(* CoDeSys 2.3.9.37 project: Cap6_10.pro *)
(* Libraries: Standard.LIB 4.10.05 12:14:46 *)

(* Global variable list: Global_Variables *)
VAR_GLOBAL

(* Entradas *)
     A:BOOL;
     B:BOOL;
     Encendido:BOOL;

(*Salidas *)
  Bomba1:BOOL;
  Bomba2:BOOL;

END_VAR

(* POU PLC_PRG, ST *)
PROGRAM PLC_PRG
VAR

END_VAR
Control();
Simulacion();
END_PROGRAM

(* POU Control, LD *)
PROGRAM Control
VAR
END_VAR
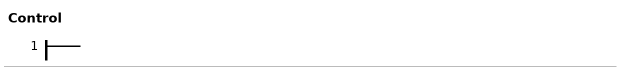
_LD_ (* Ladder Diagram *)
NETWORK 1
	*
_END_LD_
(* the same logic as Structured Text *)
(* Network 1 *)
END_PROGRAM

(* POU Simulacion, ST *)
PROGRAM Simulacion
VAR
   posy:INT;
	PrimerCiclo: BOOL:=TRUE;
	posInicial: INT;
END_VAR
IF posy>-187 THEN
IF (Bomba1=TRUE AND Bomba2=TRUE) THEN
  posy:=posy-2;
ELSE
     IF (Bomba1=TRUE OR Bomba2=TRUE) THEN
            posy:=posy-1;
     END_IF
END_IF
END_IF

IF (Bomba1=FALSE AND Bomba2=FALSE) THEN
IF posy<52 THEN
  posy:=posy+1;
END_IF
END_IF



IF posy<-50 THEN
  A:=TRUE;
ELSE
  A:=FALSE;
END_IF

IF posy<=-164 THEN
  B:=TRUE;
ELSE
  B:=FALSE;
END_IF

(* Solo en primer ciclo*)
IF (PrimerCiclo) THEN
    PrimerCiclo:=FALSE;
    posy:=posInicial;
END_IF
END_PROGRAM

(* Visualisation Deposito
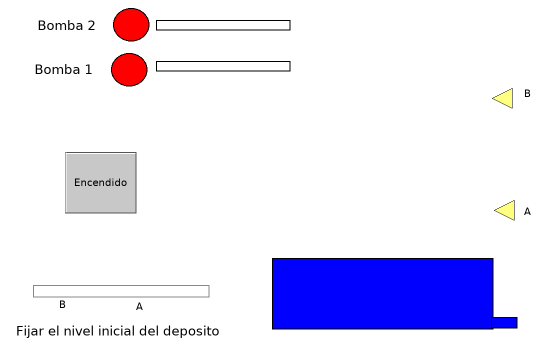
button at (94,178)-(165,239): text "Encendido"; toggles .Encendido
polygon at (521,114)-(541,134): alarm colour if .B; toggles .B
polygon at (523,226)-(543,246): alarm colour if .A; toggles .A
rectangle at (301,284)-(522,355): top Simulacion.posy
rectangle at (541,222)-(572,253): text "A"
rectangle at (541,104)-(572,135): text "B"
rectangle at (185,87)-(319,97): alarm colour if Bomba1
rectangle at (185,46)-(319,56): alarm colour if Bomba2
ellipse at (140,79)-(176,112): alarm colour if Bomba1
ellipse at (142,34)-(178,67): alarm colour if Bomba2
rectangle at (48,80)-(138,111): text "Bomba 1"
rectangle at (51,36)-(141,67): text "Bomba 2"
rectangle at (76,315)-(107,346): text "B"
rectangle at (153,317)-(184,348): text "A"
rectangle at (39,343)-(255,371): text "Fijar el nivel inicial del deposito"
4 more shapes without text or variables
*)
